{attribute 'GeneratedUsingTerminal: EPP1322-0001-0016'}
{attribute addProperty BoxType "EPP1322-0001-0016"}
{attribute addProperty Id "A_0020_EPP1322_0001_0017A_0020_EPP1322_0001_0017_8B5C362C378"}
{attribute addProperty CRC "2886107842"}
{attribute addProperty Size "378"}
TYPE A_0019_EPP1322_0001_0016_AC0682C2 EXTENDS EPP1322_AB5A9467 :
STRUCT
	{attribute addProperty Name "A_0020_EPP1322_0001_0017"}
	{attribute addProperty PreviousPort "A_0019(EPP1322-0001-0016) : D"}
	A_0020_EPP1322_0001_0017 : A_0020_EPP1322_0001_0017_8B5C362C;
END_STRUCT
END_TYPE

(* stored: Version 1.2.0.0, ProductVersion 3.1.4024.9
   DUT A_0019_EPP1322_0001_0016_AC0682C2: Id {361648b7-a693-40d5-a897-d05ddde57acc} *)
